{attribute 'linkalways'} 
{attribute 'no_explicit_call' := 'This FB is a CLASS and must be accessed using methods or properties'}
{attribute 'enable_dynamic_creation'}
FUNCTION_BLOCK Node_F_VN_AppendToContainer_TcVnRectangle_DINT EXTENDS VisionNode
VAR
    stElement : _TcVnRectangle_DINT;
    ipContainer : _ITcVnContainer;
    hrPrev : _HRESULT(S_OK);
	hresult : _HRESULT(S_OK);
END_VAR

METHOD PUBLIC  Clone : I_Node
VAR
	pNode : POINTER TO Node_F_VN_AppendToContainer_TcVnRectangle_DINT;
END_VAR
pNode := __NEW(Node_F_VN_AppendToContainer_TcVnRectangle_DINT);
Clone := pNode^;
END_METHOD

METHOD FB_init : BOOL
VAR_INPUT
	bInitRetains : BOOL; // if TRUE, the retain variables are initialized (warm start / cold start)
	bInCopyCode : BOOL;  // if TRUE, the instance afterwards gets moved into the copy code (online change)
END_VAR
AddInput('stElement', stElement);
AddInput('ipContainer', ipContainer);
AddInput('hrPrev', hrPrev);
AddOutput('ipContainer', ipContainer);
AddOutput('hresult',hresult);
END_METHOD

METHOD PROTECTED OnExecute : HRESULT
hresult.Value := F_VN_AppendToContainer_TcVnRectangle_DINT(
    stElement := stElement.Value,
	ipContainer := ipContainer.Value,
	hrPrev:= hrPrev.Value);
END_METHOD

METHOD PUBLIC PreExecutionCheck
VAR_INPUT
	Check : I_PreExecutionChecks;
END_VAR
Check.IsTrue(ipContainer.IsValid, 'ipContainer must be a valid container');
END_METHOD

END_FUNCTION_BLOCK

(* stored: Version 1.1.0.1, ProductVersion 3.1.4024.13
   POU Node_F_VN_AppendToContainer_TcVnRectangle_DINT: Id {dcbf99d1-ffd3-4548-815f-a81e0ab7372c}, SpecialFunc None
   Folder Constructor: Id {f4b6daef-871e-4554-9ca3-fab78e5174d6}
   Method Clone: Id {58343a6d-41ba-4d68-a7a8-18d908c961e9}
   Method FB_init: Id {f60de788-b934-4dad-a394-c6e67369c621}
   Method OnExecute: Id {f64740cd-675d-401d-a602-d516cbee4d54}
   Method PreExecutionCheck: Id {9d5359e8-b189-42b4-afdf-e2c381e84e66} *)
